// TIA Portal V16 export
// export: Created 2024-05-10T06:46:41.3801888Z, ExportSetting WithDefaults, DisplayName Totally Integrated Automation Portal, DisplayVersion V16, DisplayName TIA Portal Version Control Interface, DisplayVersion V16, DisplayName TIA Portal Openness, DisplayVersion V16, DisplayName STEP 7 Professional, DisplayVersion V16, DisplayName STEP 7 Safety, DisplayVersion V16, DisplayName WinCC Professional, DisplayVersion V16
FUNCTION_BLOCK "K08_指示灯"   // FB8, LAD
{ S7_Optimized_Access := 'TRUE' }
VERSION : 0.1
// stored: AutoNumber false, IsIECCheckEnabled false, IsRetainMemResEnabled false, MemoryReserve 100, SetENOAutomatically false, UDAEnableTagReadback false
BEGIN

REGION Network 1: 自动灯
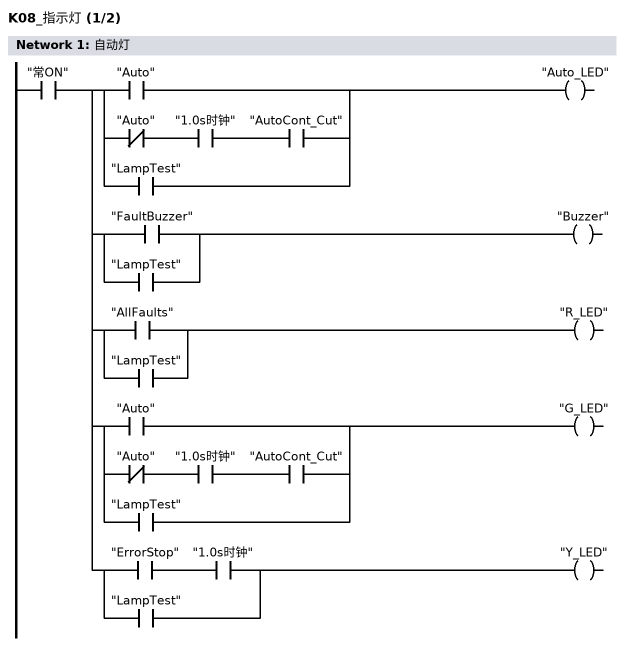
   RUNG wire#powerrail
      Contact( "常ON" )
      wire#w1
      Contact( "Auto" )
      wire#w2
      Coil( "Auto_LED" )
   END_RUNG
   RUNG wire#w1
      I_Contact( "Auto" )
      Contact( "1.0s时钟" )
      Contact( "AutoCont_Cut" )
   END_RUNG wire#w2
   RUNG wire#w1
      Contact( "LampTest" )
   END_RUNG wire#w2
   RUNG wire#w1
      Contact( "FaultBuzzer" )
      wire#w3
      Coil( "Buzzer" )
   END_RUNG
   RUNG wire#w1
      Contact( "LampTest" )
   END_RUNG wire#w3
   RUNG wire#w1
      Contact( "AllFaults" )
      wire#w4
      Coil( "R_LED" )
   END_RUNG
   RUNG wire#w1
      Contact( "LampTest" )
   END_RUNG wire#w4
   RUNG wire#w1
      Contact( "Auto" )
      wire#w5
      Coil( "G_LED" )
   END_RUNG
   RUNG wire#w1
      I_Contact( "Auto" )
      Contact( "1.0s时钟" )
      Contact( "AutoCont_Cut" )
   END_RUNG wire#w5
   RUNG wire#w1
      Contact( "LampTest" )
   END_RUNG wire#w5
   RUNG wire#w1
      Contact( "ErrorStop" )
      Contact( "1.0s时钟" )
      wire#w6
      Coil( "Y_LED" )
   END_RUNG
   RUNG wire#w1
      Contact( "LampTest" )
   END_RUNG wire#w6
   // the same network as SCL:
   "Auto_LED" := "常ON" AND ("Auto" OR (NOT "Auto" AND "1.0s时钟" AND "AutoCont_Cut") OR "LampTest");
   "Buzzer" := "常ON" AND ("FaultBuzzer" OR "LampTest");
   "R_LED" := "常ON" AND ("AllFaults" OR "LampTest");
   "G_LED" := "常ON" AND ("Auto" OR (NOT "Auto" AND "1.0s时钟" AND "AutoCont_Cut") OR "LampTest");
   "Y_LED" := "常ON" AND (("ErrorStop" AND "1.0s时钟") OR "LampTest");
END_REGION

REGION Network 2: 放行灯
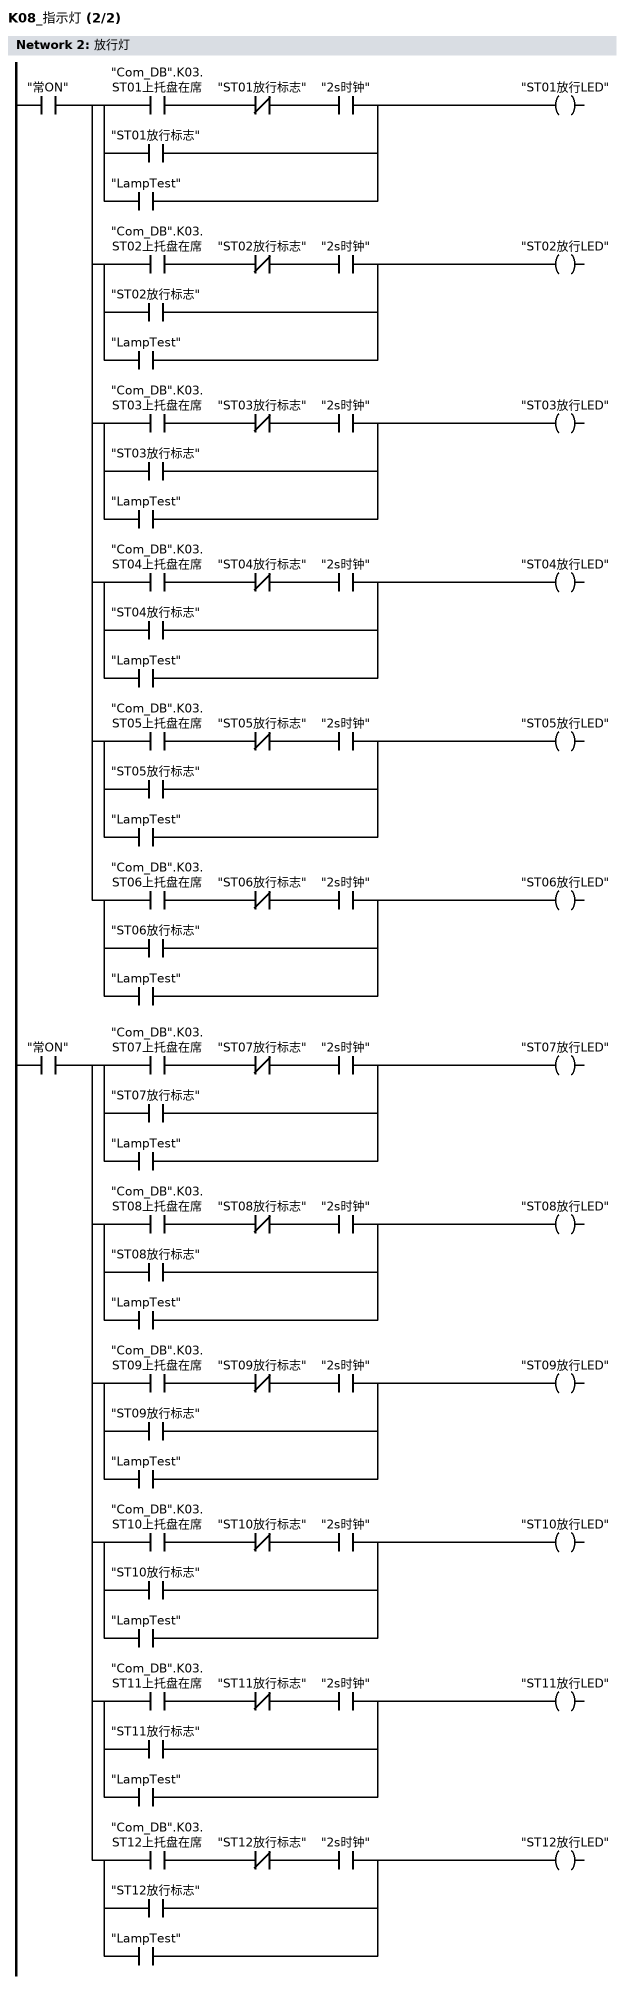
   RUNG wire#powerrail
      Contact( "常ON" )
      wire#w1
      Contact( "Com_DB".K03.ST01上托盘在席 )
      I_Contact( "ST01放行标志" )
      Contact( "2s时钟" )
      wire#w2
      Coil( "ST01放行LED" )
   END_RUNG
   RUNG wire#w1
      Contact( "ST01放行标志" )
   END_RUNG wire#w2
   RUNG wire#w1
      Contact( "LampTest" )
   END_RUNG wire#w2
   RUNG wire#w1
      Contact( "Com_DB".K03.ST02上托盘在席 )
      I_Contact( "ST02放行标志" )
      Contact( "2s时钟" )
      wire#w3
      Coil( "ST02放行LED" )
   END_RUNG
   RUNG wire#w1
      Contact( "ST02放行标志" )
   END_RUNG wire#w3
   RUNG wire#w1
      Contact( "LampTest" )
   END_RUNG wire#w3
   RUNG wire#w1
      Contact( "Com_DB".K03.ST03上托盘在席 )
      I_Contact( "ST03放行标志" )
      Contact( "2s时钟" )
      wire#w4
      Coil( "ST03放行LED" )
   END_RUNG
   RUNG wire#w1
      Contact( "ST03放行标志" )
   END_RUNG wire#w4
   RUNG wire#w1
      Contact( "LampTest" )
   END_RUNG wire#w4
   RUNG wire#w1
      Contact( "Com_DB".K03.ST04上托盘在席 )
      I_Contact( "ST04放行标志" )
      Contact( "2s时钟" )
      wire#w5
      Coil( "ST04放行LED" )
   END_RUNG
   RUNG wire#w1
      Contact( "ST04放行标志" )
   END_RUNG wire#w5
   RUNG wire#w1
      Contact( "LampTest" )
   END_RUNG wire#w5
   RUNG wire#w1
      Contact( "Com_DB".K03.ST05上托盘在席 )
      I_Contact( "ST05放行标志" )
      Contact( "2s时钟" )
      wire#w6
      Coil( "ST05放行LED" )
   END_RUNG
   RUNG wire#w1
      Contact( "ST05放行标志" )
   END_RUNG wire#w6
   RUNG wire#w1
      Contact( "LampTest" )
   END_RUNG wire#w6
   RUNG wire#w1
      Contact( "Com_DB".K03.ST06上托盘在席 )
      I_Contact( "ST06放行标志" )
      Contact( "2s时钟" )
      wire#w7
      Coil( "ST06放行LED" )
   END_RUNG
   RUNG wire#w1
      Contact( "ST06放行标志" )
   END_RUNG wire#w7
   RUNG wire#w1
      Contact( "LampTest" )
   END_RUNG wire#w7
   RUNG wire#powerrail
      Contact( "常ON" )
      wire#w8
      Contact( "Com_DB".K03.ST07上托盘在席 )
      I_Contact( "ST07放行标志" )
      Contact( "2s时钟" )
      wire#w9
      Coil( "ST07放行LED" )
   END_RUNG
   RUNG wire#w8
      Contact( "ST07放行标志" )
   END_RUNG wire#w9
   RUNG wire#w8
      Contact( "LampTest" )
   END_RUNG wire#w9
   RUNG wire#w8
      Contact( "Com_DB".K03.ST08上托盘在席 )
      I_Contact( "ST08放行标志" )
      Contact( "2s时钟" )
      wire#w10
      Coil( "ST08放行LED" )
   END_RUNG
   RUNG wire#w8
      Contact( "ST08放行标志" )
   END_RUNG wire#w10
   RUNG wire#w8
      Contact( "LampTest" )
   END_RUNG wire#w10
   RUNG wire#w8
      Contact( "Com_DB".K03.ST09上托盘在席 )
      I_Contact( "ST09放行标志" )
      Contact( "2s时钟" )
      wire#w11
      Coil( "ST09放行LED" )
   END_RUNG
   RUNG wire#w8
      Contact( "ST09放行标志" )
   END_RUNG wire#w11
   RUNG wire#w8
      Contact( "LampTest" )
   END_RUNG wire#w11
   RUNG wire#w8
      Contact( "Com_DB".K03.ST10上托盘在席 )
      I_Contact( "ST10放行标志" )
      Contact( "2s时钟" )
      wire#w12
      Coil( "ST10放行LED" )
   END_RUNG
   RUNG wire#w8
      Contact( "ST10放行标志" )
   END_RUNG wire#w12
   RUNG wire#w8
      Contact( "LampTest" )
   END_RUNG wire#w12
   RUNG wire#w8
      Contact( "Com_DB".K03.ST11上托盘在席 )
      I_Contact( "ST11放行标志" )
      Contact( "2s时钟" )
      wire#w13
      Coil( "ST11放行LED" )
   END_RUNG
   RUNG wire#w8
      Contact( "ST11放行标志" )
   END_RUNG wire#w13
   RUNG wire#w8
      Contact( "LampTest" )
   END_RUNG wire#w13
   RUNG wire#w8
      Contact( "Com_DB".K03.ST12上托盘在席 )
      I_Contact( "ST12放行标志" )
      Contact( "2s时钟" )
      wire#w14
      Coil( "ST12放行LED" )
   END_RUNG
   RUNG wire#w8
      Contact( "ST12放行标志" )
   END_RUNG wire#w14
   RUNG wire#w8
      Contact( "LampTest" )
   END_RUNG wire#w14
   // the same network as SCL:
   "ST01放行LED" := "常ON" AND (("Com_DB".K03.ST01上托盘在席 AND NOT "ST01放行标志" AND "2s时钟") OR "ST01放行标志" OR "LampTest");
   "ST02放行LED" := "常ON" AND (("Com_DB".K03.ST02上托盘在席 AND NOT "ST02放行标志" AND "2s时钟") OR "ST02放行标志" OR "LampTest");
   "ST03放行LED" := "常ON" AND (("Com_DB".K03.ST03上托盘在席 AND NOT "ST03放行标志" AND "2s时钟") OR "ST03放行标志" OR "LampTest");
   "ST04放行LED" := "常ON" AND (("Com_DB".K03.ST04上托盘在席 AND NOT "ST04放行标志" AND "2s时钟") OR "ST04放行标志" OR "LampTest");
   "ST05放行LED" := "常ON" AND (("Com_DB".K03.ST05上托盘在席 AND NOT "ST05放行标志" AND "2s时钟") OR "ST05放行标志" OR "LampTest");
   "ST06放行LED" := "常ON" AND (("Com_DB".K03.ST06上托盘在席 AND NOT "ST06放行标志" AND "2s时钟") OR "ST06放行标志" OR "LampTest");
   "ST07放行LED" := "常ON" AND (("Com_DB".K03.ST07上托盘在席 AND NOT "ST07放行标志" AND "2s时钟") OR "ST07放行标志" OR "LampTest");
   "ST08放行LED" := "常ON" AND (("Com_DB".K03.ST08上托盘在席 AND NOT "ST08放行标志" AND "2s时钟") OR "ST08放行标志" OR "LampTest");
   "ST09放行LED" := "常ON" AND (("Com_DB".K03.ST09上托盘在席 AND NOT "ST09放行标志" AND "2s时钟") OR "ST09放行标志" OR "LampTest");
   "ST10放行LED" := "常ON" AND (("Com_DB".K03.ST10上托盘在席 AND NOT "ST10放行标志" AND "2s时钟") OR "ST10放行标志" OR "LampTest");
   "ST11放行LED" := "常ON" AND (("Com_DB".K03.ST11上托盘在席 AND NOT "ST11放行标志" AND "2s时钟") OR "ST11放行标志" OR "LampTest");
   "ST12放行LED" := "常ON" AND (("Com_DB".K03.ST12上托盘在席 AND NOT "ST12放行标志" AND "2s时钟") OR "ST12放行标志" OR "LampTest");
END_REGION
END_FUNCTION_BLOCK
